// TIA Portal V19 export
FUNCTION "LAF_ReadPlcDateAndTime" : Void   // FC19, LAD
TITLE = LAF_ReadPlcDateAndTime
AUTHOR : Siemens Digital Industries
FAMILY : LAF
VERSION : 1.2
// This blocks reads the current local time of the PLC and provides it in different formats.
// stored: Access Published, IsIECCheckEnabled true, SetENOAutomatically false
   VAR_IN_OUT
      currentDateAndTime : "LAF_typeGlobalDateTime";
   END_VAR
BEGIN

REGION Network 1: BLOCK INFO HEADER
   // SIEMENS AG / (c)Copyright 2024
   // ------------------------------------------------------------------------------
   // Title:            LAF_ReadPlcDataAndTime
   // Comment/Function: This blocks reads the current local time of the PLC and provides it in different formats.
   // Library/Family:   Library of Automation Framework
   // Author:                Siemens Digital Industry
   // Tested with:       S7-PLCSIM Advanced 6.0
   // Engineering:      TIA Portal V19
   // Restrictions:       ---
   // Requirements:   ---
   // ------------------------------------------------------------------------------
   // Change log table:
   // Version  | Date       | Expert in charge       | Changes applied
   // ---------|------------|------------------------|------------------------------
   // 01.01.00 | 21.06.2024 | SIMATIC Systems Support
   //                         First released version
   // 01.02.00 | 30.09.2024 | SIMATIC Systems Support
   //                         Block information properties updated
END_REGION

REGION Network 2: DESCRIPTION
   // This block reads the system's local time and then converts it into two additional different formats (_LDT_ and _Date_And_Time_) for subsequent use in the program.
END_REGION

REGION Network 3: Read local time / SPS: Datum & Uhrzeit
   // Verwaltung von Datum und Uhrzeit der SPS. Konvertiergung dieser in verschiedene Formate und zuweisung auf den InOut Parameter
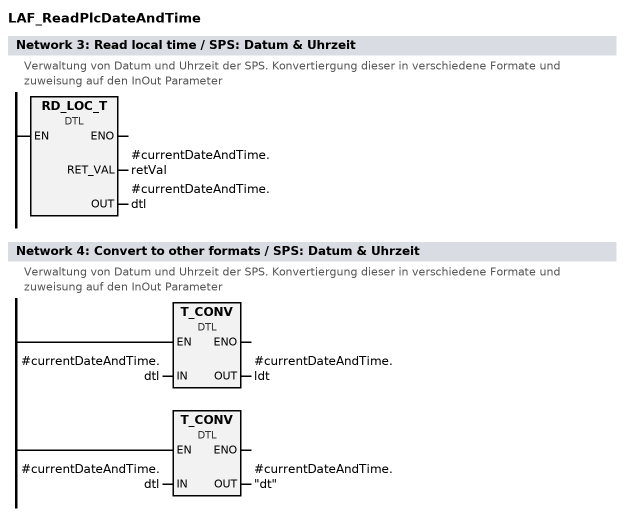
   RUNG wire#powerrail
      { S7_Templates := "date_type := DTL" } RD_LOC_T(RET_VAL => #currentDateAndTime.retVal, OUT => #currentDateAndTime.dtl)
   END_RUNG
   // the same network as SCL:
   #currentDateAndTime.retVal := RD_LOC_T(OUT => #currentDateAndTime.dtl);
END_REGION

REGION Network 4: Convert to other formats / SPS: Datum & Uhrzeit
   // Verwaltung von Datum und Uhrzeit der SPS. Konvertiergung dieser in verschiedene Formate und zuweisung auf den InOut Parameter
   RUNG wire#powerrail
      { S7_Templates := "[src_type := DTL, dest_type := LDT]" } T_CONV(IN := #currentDateAndTime.dtl, OUT => #currentDateAndTime.ldt)
   END_RUNG
   RUNG wire#powerrail
      { S7_Templates := "[src_type := DTL, dest_type := Date_And_Time]" } T_CONV(IN := #currentDateAndTime.dtl, OUT => #currentDateAndTime."dt")
   END_RUNG
   // the same network as SCL:
   T_CONV(IN := #currentDateAndTime.dtl, OUT => #currentDateAndTime.ldt);
   T_CONV(IN := #currentDateAndTime.dtl, OUT => #currentDateAndTime."dt");
END_REGION
END_FUNCTION
